FUNCTION_BLOCK TempRoomWithMultipleSensors
VAR_GENERIC CONSTANT
	SENSOR_CAP		: UDINT := 4;
END_VAR
IMPLEMENTS I_Execute
VAR CONSTANT
	STATE_CAP		: UDINT := 5;
END_VAR
VAR
	_this			: Entity;
	_ctx			: Room_Ctx;
	_room			: RoomInterface(_ctx);
	_tag			: Tag(CONCAT('Room_', UDINT_TO_STRING(_room.Id)));
	_compTag		: Comp(_tag, _this);
	_exe			: Execute(THIS^);
	
	_uiLogic		: Room_UiLogic(_ctx);
	
	_systemReceiver	: Room_SystemReceiver(_ctx);
	
	_smgr			: StateManager<STATE_CAP>(_this);
	_proxSmgr		: StateManagerProxy(_smgr, _ctx.state.iMgr);
	
	_disable		: Room_State_Disabled(_this, _ctx);
	_proxDisable	: StateProxy(_disable, _ctx.state.iDisable);
	
	_fault			: Room_State_Fault(_this,_ctx);
	_proxFault		: StateProxy(_fault, _ctx.state.iFault);	
	
	_idle			: Room_State_Idle(_this,_ctx);
	_proxIdle		: StateProxy(_idle, _ctx.state.iIdle);	
	
	_systemOff		: Room_State_SystemOff(_this,_ctx);
	_proxSystemOff	: StateProxy(_systemOff, _ctx.state.iSystemOff);
END_VAR

	// Here add custom components

VAR PERSISTENT
	_settings				: Room_Settings_TemperatureSettings;
END_VAR
VAR_INPUT
	rTemperature			: ARRAY[1..SENSOR_CAP] OF REAL;
	
	bInletValveIsOpen		: BOOL;
	bInletValveIsClosed		: BOOL;
	
	bOutletValveIsOpen		: BOOL;
	bOutletValveIsClosed	: BOOL;
END_VAR
VAR
	_rTemperature			: REAL;
END_VAR
VAR_OUTPUT
	bInletValve				: BOOL;
	bOutletValve			: BOOL;
END_VAR
VAR
	_tempDemand		: Room_State_DemandTemperature(_this, _ctx, _settings, _rTemperature);
END_VAR

METHOD Execute
VAR
	i			: UDINT;
	_rTempSum	: REAL;
END_VAR
_ctx.priv.bClosed := bInletValveIsClosed AND bOutletValveIsClosed;
_ctx.priv.bOpen := bInletValveIsOpen AND bOutletValveIsOpen;

bInletValve :=  _ctx.io.bOpenValves;
bOutletValve :=  _ctx.io.bOpenValves;

FOR i := 1 TO SENSOR_CAP DO
	_rTempSum := rTemperature[i] + _rTempSum;
END_FOR

_rTemperature := _rTempSum/UDINT_TO_REAL(SENSOR_CAP);
END_METHOD

END_FUNCTION_BLOCK

(* stored: Version 1.1.0.1
   POU TempRoomWithMultipleSensors: Id {1c1f35f1-e452-44bd-ba56-2c114335a3d0}, SpecialFunc None
   Method Execute: Id {227dadc6-9c24-4539-890a-d7ee861363ab} *)
